FUNCTION FUN_ConvOneByteToInt8 : INT
VAR_INPUT
	nValue1		:BYTE;				// Input Byte no 1

END_VAR
VAR
	uData		:U_Convert_INT8;		// Data variable used for conversion
END_VAR

// Save input bytes in data union
uData.nBYTE := nValue1;


// Return value
FUN_ConvOneByteToInt8 := uData.nValue;

END_FUNCTION

(* stored: Version 1.1.0.1, ProductVersion 3.1.4024.12
   POU FUN_ConvOneByteToInt8: Id {f828b272-e539-4f8d-9b4b-d0b5524e0d05}, SpecialFunc None *)
